Staubli VAL3: init.pgx

program init()
  local num l_nLink
  local num l_nNum
begin
  //variables
  bPause=false
  bExit=false
  bForceError=false
  bTableAlm=false
  bSuspend=false
  bUpload=false

  bInterVal=false
  for l_nNum=0 to 5
    bRefreshMsg[l_nNum]=true
  endFor
  //
  read:bCycle=false
  //转台转动与否
  date:bWorTbMoving=false
  //IO
  call io:init()
  call io:tableSpeed(nTabSpeed)
  //init ATI
  call ati:initialize("io:sAtiFs",l_nLink)
end
